(* LS Electric XG5000 project: AA_BB_ *)
(* PLC LSPLC *)
VAR_GLOBAL
    Flag_1 : BOOL;
    flag_2 : BOOL;
    flag_3 : BOOL;
    Relay_1 AT %QX0.0.1 : BOOL;
    Relay_2 AT %QX0.0.2 : BOOL;
    Sensor_1 AT %IX0.0.1 : BOOL;
    Sensor_2 AT %IX0.0.2 : BOOL;
    Sensor_3 AT %IX0.0.3 : BOOL;
    Sensor_4 AT %IX0.0.4 : BOOL;
END_VAR

PROGRAM NewProgram (* task: Scan Program *)
VAR_EXTERNAL
    Flag_1 : BOOL;
    flag_2 : BOOL;
    flag_3 : BOOL;
    Relay_1 : BOOL; (* AT %QX0.0.1 *)
    Relay_2 : BOOL; (* AT %QX0.0.2 *)
    Sensor_1 : BOOL; (* AT %IX0.0.1 *)
    Sensor_2 : BOOL; (* AT %IX0.0.2 *)
    Sensor_3 : BOOL; (* AT %IX0.0.3 *)
    Sensor_4 : BOOL; (* AT %IX0.0.4 *)
END_VAR

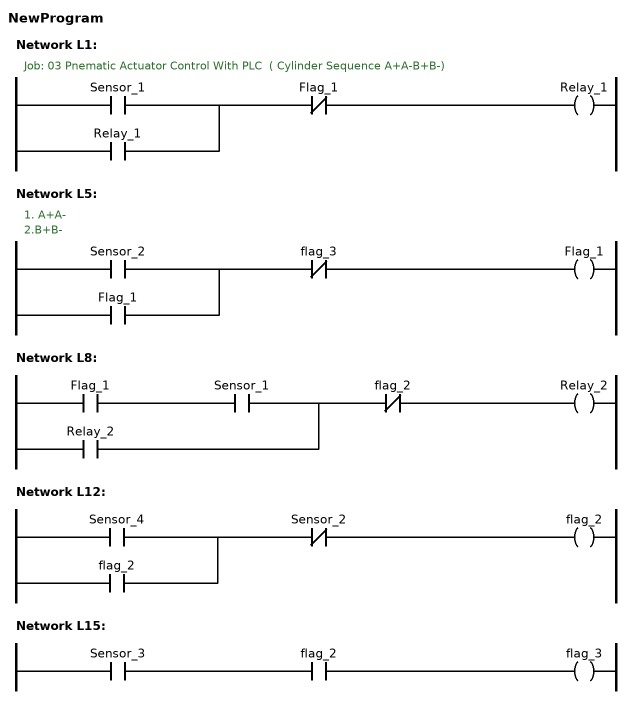
(* Job: 03 Pnematic Actuator Control With PLC  ( Cylinder Sequence A+A-B+B-) *)
(* Rung L1 *)
Relay_1 := (Sensor_1 OR Relay_1) AND NOT Flag_1;
(* 1. A+A- *)
(* 2.B+B- *)
(* Rung L5 *)
Flag_1 := (Sensor_2 OR Flag_1) AND NOT flag_3;
(* Rung L8 *)
Relay_2 := ((Flag_1 AND Sensor_1) OR Relay_2) AND NOT flag_2;
(* Rung L12 *)
flag_2 := (Sensor_4 OR flag_2) AND NOT Sensor_2;
(* Rung L15 *)
flag_3 := Sensor_3 AND flag_2;
END_PROGRAM